SYSTEM Read_Write_Remote_Server
  (* Version 1.0, 2025-01-17, Bruno *)
  APPLICATION Read_Write_Remote_ServerApp
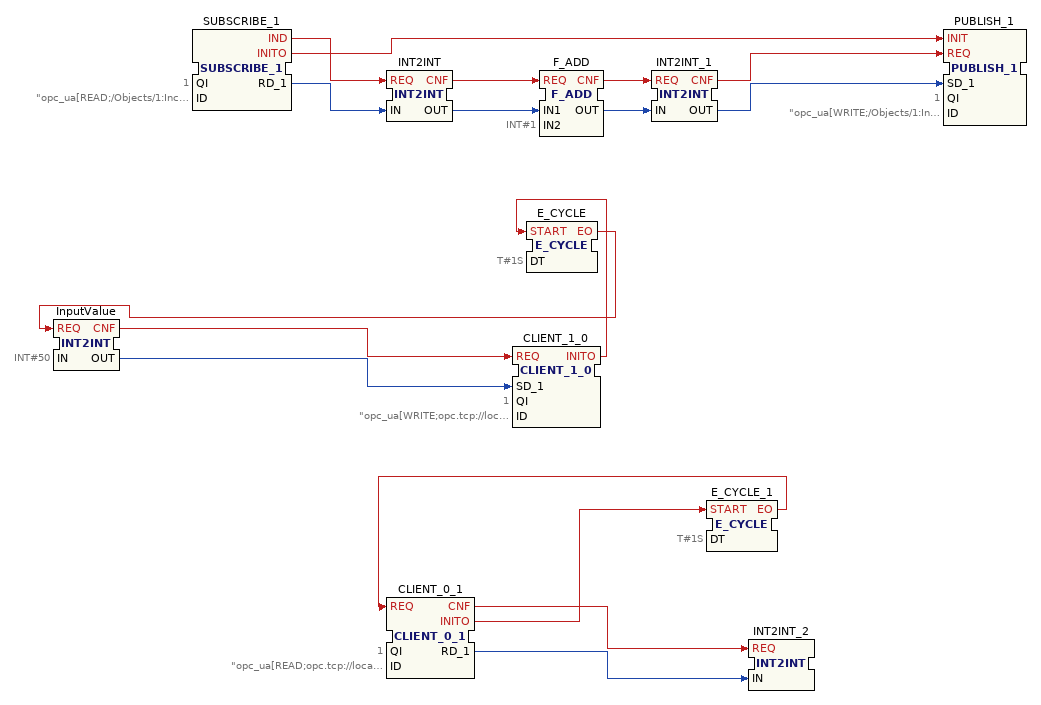
    FBS
      SUBSCRIBE_1 : SUBSCRIBE_1(QI := 1, ID := "opc_ua[READ;/Objects/1:Incrementer]");
      PUBLISH_1 : PUBLISH_1(QI := 1, ID := "opc_ua[WRITE;/Objects/1:Incremented]");
      INT2INT : INT2INT;
      F_ADD : F_ADD(IN2 := INT#1);
      INT2INT_1 : INT2INT;
      CLIENT_1_0 : CLIENT_1_0(QI := 1, ID := "opc_ua[WRITE;opc.tcp://localhost:4840#;/Objects/1:Incrementer]");
      InputValue : INT2INT(IN := INT#50);
      E_CYCLE : E_CYCLE(DT := T#1S);
      INT2INT_2 : INT2INT;
      CLIENT_0_1 : CLIENT_0_1(QI := 1, ID := "opc_ua[READ;opc.tcp://localhost:4840#;/Objects/1:Incremented]");
      E_CYCLE_1 : E_CYCLE(DT := T#1S);
    END_FBS
    EVENT_CONNECTIONS
      SUBSCRIBE_1.IND TO INT2INT.REQ;
      SUBSCRIBE_1.INITO TO PUBLISH_1.INIT;
      INT2INT.CNF TO F_ADD.REQ;
      F_ADD.CNF TO INT2INT_1.REQ;
      INT2INT_1.CNF TO PUBLISH_1.REQ;
      InputValue.CNF TO CLIENT_1_0.REQ;
      CLIENT_1_0.INITO TO E_CYCLE.START;
      E_CYCLE.EO TO InputValue.REQ;
      CLIENT_0_1.CNF TO INT2INT_2.REQ;
      CLIENT_0_1.INITO TO E_CYCLE_1.START;
      E_CYCLE_1.EO TO CLIENT_0_1.REQ;
    END_CONNECTIONS
    DATA_CONNECTIONS
      SUBSCRIBE_1.RD_1 TO INT2INT.IN;
      INT2INT.OUT TO F_ADD.IN1;
      F_ADD.OUT TO INT2INT_1.IN;
      INT2INT_1.OUT TO PUBLISH_1.SD_1;
      InputValue.OUT TO CLIENT_1_0.SD_1;
      CLIENT_0_1.RD_1 TO INT2INT_2.IN;
    END_CONNECTIONS
  END_APPLICATION
  DEVICE FORTE_Server : FORTE_PC(MGR_ID := "localhost:61499")
    {SET_ATTRIBUTE(Profile, HOLOBLOC)} (* device profile *)
    RESOURCE EMB_RES : EMB_RES
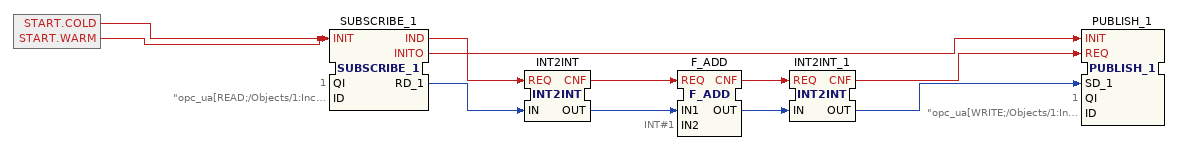
      FBS
        SUBSCRIBE_1 : SUBSCRIBE_1(QI := 1, ID := "opc_ua[READ;/Objects/1:Incrementer]");
        INT2INT : INT2INT;
        F_ADD : F_ADD(IN2 := INT#1);
        INT2INT_1 : INT2INT;
        PUBLISH_1 : PUBLISH_1(QI := 1, ID := "opc_ua[WRITE;/Objects/1:Incremented]");
      END_FBS
      EVENT_CONNECTIONS
        SUBSCRIBE_1.IND TO INT2INT.REQ;
        INT2INT.CNF TO F_ADD.REQ;
        F_ADD.CNF TO INT2INT_1.REQ;
        SUBSCRIBE_1.INITO TO PUBLISH_1.INIT;
        INT2INT_1.CNF TO PUBLISH_1.REQ;
        START.COLD TO SUBSCRIBE_1.INIT;
        START.WARM TO SUBSCRIBE_1.INIT;
      END_CONNECTIONS
      DATA_CONNECTIONS
        SUBSCRIBE_1.RD_1 TO INT2INT.IN;
        INT2INT.OUT TO F_ADD.IN1;
        F_ADD.OUT TO INT2INT_1.IN;
        INT2INT_1.OUT TO PUBLISH_1.SD_1;
      END_CONNECTIONS
    END_RESOURCE
  END_DEVICE
  DEVICE FORTE_Client : FORTE_PC(MGR_ID := "localhost:61500")
    {SET_ATTRIBUTE(Profile, HOLOBLOC)} (* device profile *)
    RESOURCE EMB_RES : EMB_RES
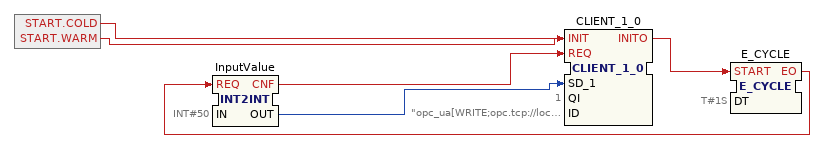
      FBS
        CLIENT_1_0 : CLIENT_1_0(QI := 1, ID := "opc_ua[WRITE;opc.tcp://localhost:4840#;/Objects/1:Incrementer]");
        InputValue : INT2INT(IN := INT#50);
        E_CYCLE : E_CYCLE(DT := T#1S);
      END_FBS
      EVENT_CONNECTIONS
        START.COLD TO CLIENT_1_0.INIT;
        START.WARM TO CLIENT_1_0.INIT;
        InputValue.CNF TO CLIENT_1_0.REQ;
        CLIENT_1_0.INITO TO E_CYCLE.START;
        E_CYCLE.EO TO InputValue.REQ;
      END_CONNECTIONS
      DATA_CONNECTIONS
        InputValue.OUT TO CLIENT_1_0.SD_1;
      END_CONNECTIONS
    END_RESOURCE
  END_DEVICE
  DEVICE FORTE_PC_Client1 : FORTE_PC(MGR_ID := "localhost:61501")
    {SET_ATTRIBUTE(Profile, HOLOBLOC)} (* device profile *)
    RESOURCE EMB_RES : EMB_RES
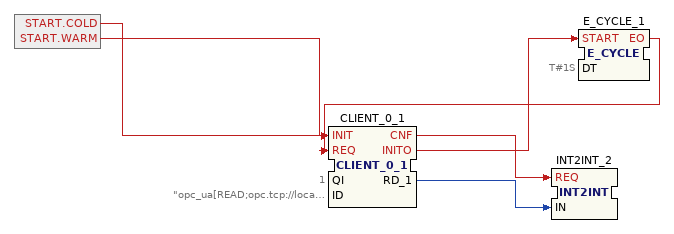
      FBS
        INT2INT_2 : INT2INT;
        CLIENT_0_1 : CLIENT_0_1(QI := 1, ID := "opc_ua[READ;opc.tcp://localhost:4840#;/Objects/1:Incremented]");
        E_CYCLE_1 : E_CYCLE(DT := T#1S);
      END_FBS
      EVENT_CONNECTIONS
        CLIENT_0_1.CNF TO INT2INT_2.REQ;
        START.COLD TO CLIENT_0_1.INIT;
        START.WARM TO CLIENT_0_1.INIT;
        CLIENT_0_1.INITO TO E_CYCLE_1.START;
        E_CYCLE_1.EO TO CLIENT_0_1.REQ;
      END_CONNECTIONS
      DATA_CONNECTIONS
        CLIENT_0_1.RD_1 TO INT2INT_2.IN;
      END_CONNECTIONS
    END_RESOURCE
  END_DEVICE
  MAPPINGS
    Read_Write_Remote_ServerApp.SUBSCRIBE_1 ON FORTE_Server.EMB_RES.SUBSCRIBE_1;
    Read_Write_Remote_ServerApp.INT2INT ON FORTE_Server.EMB_RES.INT2INT;
    Read_Write_Remote_ServerApp.F_ADD ON FORTE_Server.EMB_RES.F_ADD;
    Read_Write_Remote_ServerApp.INT2INT_1 ON FORTE_Server.EMB_RES.INT2INT_1;
    Read_Write_Remote_ServerApp.PUBLISH_1 ON FORTE_Server.EMB_RES.PUBLISH_1;
    Read_Write_Remote_ServerApp.CLIENT_1_0 ON FORTE_Client.EMB_RES.CLIENT_1_0;
    Read_Write_Remote_ServerApp.InputValue ON FORTE_Client.EMB_RES.InputValue;
    Read_Write_Remote_ServerApp.E_CYCLE ON FORTE_Client.EMB_RES.E_CYCLE;
    Read_Write_Remote_ServerApp.INT2INT_2 ON FORTE_PC_Client1.EMB_RES.INT2INT_2;
    Read_Write_Remote_ServerApp.CLIENT_0_1 ON FORTE_PC_Client1.EMB_RES.CLIENT_0_1;
    Read_Write_Remote_ServerApp.E_CYCLE_1 ON FORTE_PC_Client1.EMB_RES.E_CYCLE_1;
  END_MAPPINGS
  SEGMENTS
    Ethernet : Ethernet;
  END_SEGMENTS
  LINKS
    FORTE_Server => Ethernet;
    FORTE_Client => Ethernet;
    FORTE_PC_Client1 => Ethernet;
  END_LINKS
END_SYSTEM
